Staubli VAL3: VelocityCfg.dtx

public num nCmdType
public num nRefFrameVec[6]
public num nToolVec[6]
public num nAccel
public num nVel
public num nTransVel
public num nRotVel
